Universal Robots PolyScope program: ToolAngleStep_1.urp

ProgramRoot directory=/home/ur/ursim-3.1/programs/Support site; kinematics=(a=[0, -0.612, -0.5723, 0, 0, 0], d=[0.118, 0, 0, 0.16394, 0.1157, 0.0922], alpha=[1.5708, 0, 0, 1.5708, -1.5708, 0], deltaTheta=[0, 0, 0, 0, 0, 0], status=notInitialized); lastSavedInVersion=(project__name=Polyscope, major__version=3, minor__version=1, svn__revision=18024, build__date=Jul 07 2015, 15:18:49); name=toolAngleStep; programVersion=(project__name=Polyscope, major__version=3, minor__version=1, svn__revision=18024, build__date=Jul 07 2015, 15:18:49); robotEnvironmentFileName=default; serialNumberRobot=2015350001
  MainProgram cartesianAcceleration=1.2; cartesianSpeed=0.25; jointAcceleration=1.3962634015954636; jointSpeed=1.0471975511965976; sharedProcessMoveBlendRadius=0.025; motionType=JOINT_SPACE
    Assignment expr=get_joint_positions(); operatorValueType=INTEGER; valueSource=EXPRESSION
    Script type=0; expressionBranchNode=b[5]=b[5]+d2r(10)
    Script type=0; expressionBranchNode=movej(b)
    Wait 
    Script type=0; expressionBranchNode=b[5]=b[5]+d2r(10)
    Script type=0; expressionBranchNode=movej(b)
    Wait 
    Script type=0; expressionBranchNode=b[5]=b[5]-d2r(20)
    Script type=0; expressionBranchNode=movej(b)
    Wait 
